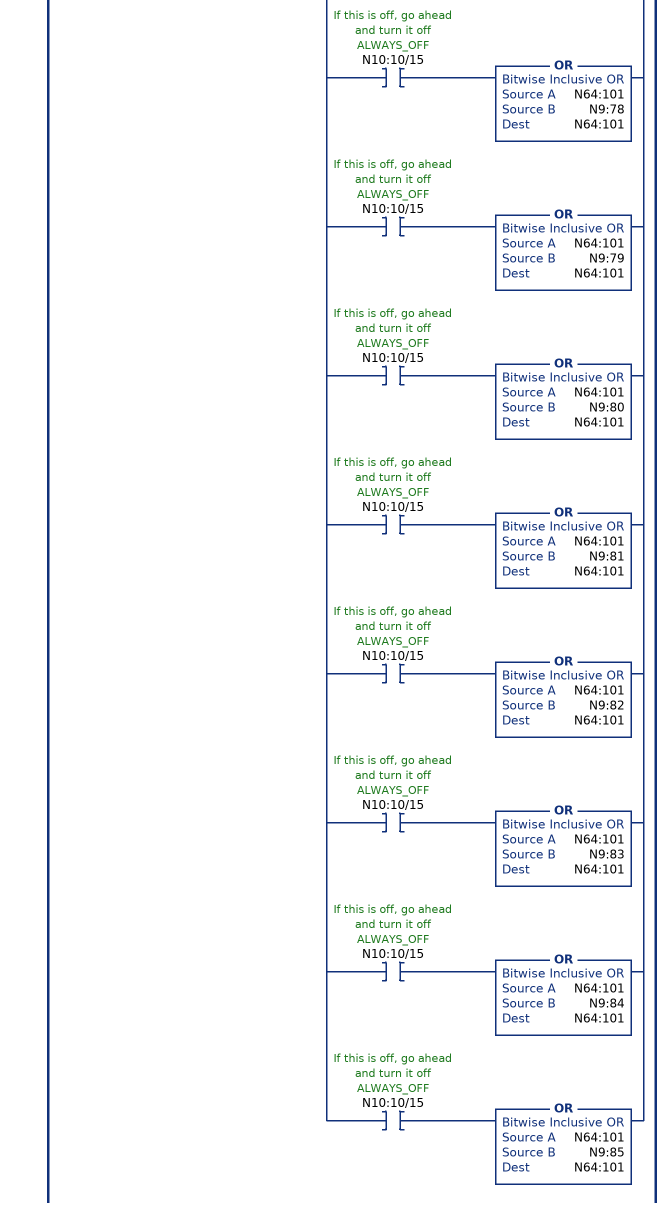
% Rung: 28 %
SOR EQU C5:19.ACC 11 XIO B3:0/3 BST MOV 0 N64:101 NXB XIC N10:10/15 OR N64:101 N9:70 N64:101 NXB XIC N10:10/15 OR N64:101 N9:71 N64:101 NXB XIC N10:10/15 OR N64:101 N9:72 N64:101 NXB XIC N10:10/15 OR N64:101 N9:73 N64:101 NXB XIC N10:10/15 OR N64:101 N9:74 N64:101 NXB XIC N10:10/15 OR N64:101 N9:75 N64:101 NXB XIC N10:10/15 OR N64:101 N9:76 N64:101 NXB XIC N10:10/15 OR N64:101 N9:77 N64:101 NXB XIC N10:10/15 OR N64:101 N9:78 N64:101 NXB XIC N10:10/15 OR N64:101 N9:79 N64:101 NXB XIC N10:10/15 OR N64:101 N9:80 N64:101 NXB XIC N10:10/15 OR N64:101 N9:81 N64:101 NXB XIC N10:10/15 OR N64:101 N9:82 N64:101 NXB XIC N10:10/15 OR N64:101 N9:83 N64:101 NXB XIC N10:10/15 OR N64:101 N9:84 N64:101 NXB XIC N10:10/15 OR N64:101 N9:85 N64:101 BND EOR
%   C5:19  MODBUS_COIL_CTR %
%   B3:0/3  MODBUS_TEST %
%   N10:10/15  ALWAYS_OFF  "If this is off, go ahead and turn it off" %
%   N9:70  BIT_0 %
%   N9:71  BIT_1 %
%   N9:72  BIT_2 %
%   N9:73  BIT_3 %
%   N9:74  BIT_4 %
%   N9:75  BIT_5 %
%   N9:76  BIT_6 %
%   N9:77  BIT_7 %
%   N9:78  BIT_8 %
%   N9:79  BIT_9 %
%   N9:80  BIT_10 %
%   N9:81  BIT_11 %
%   N9:82  BIT_12 %
%   N9:83  BIT_13 %
%   N9:84  BIT_14 %
%   N9:85  BIT_15 %

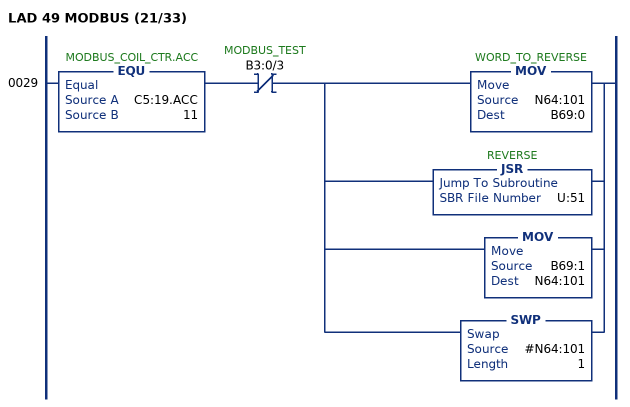
% Rung: 29 %
SOR EQU C5:19.ACC 11 XIO B3:0/3 BST MOV N64:101 B69:0 NXB JSR U:51 NXB MOV B69:1 N64:101 NXB SWP #N64:101 1 BND EOR
%   C5:19  MODBUS_COIL_CTR %
%   B3:0/3  MODBUS_TEST %
%   B69:0  WORD_TO_REVERSE %
%   U:51  REVERSE %
%   B69:1  REVERSED_WORD %

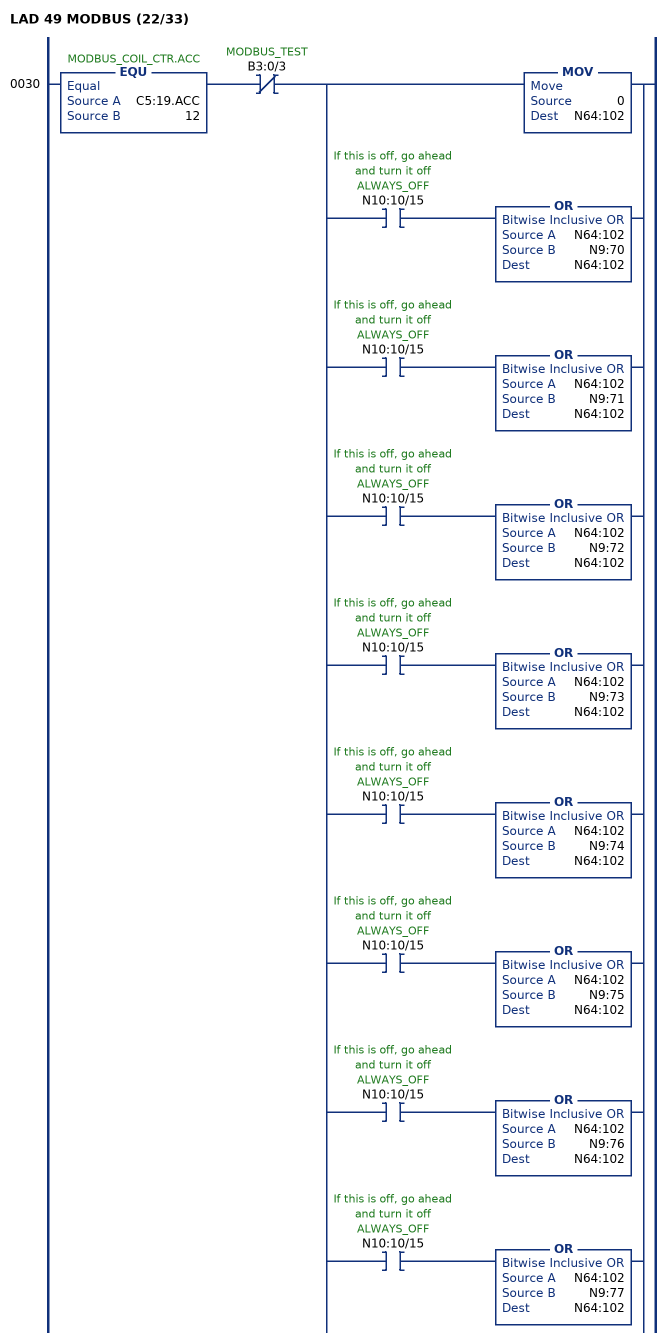

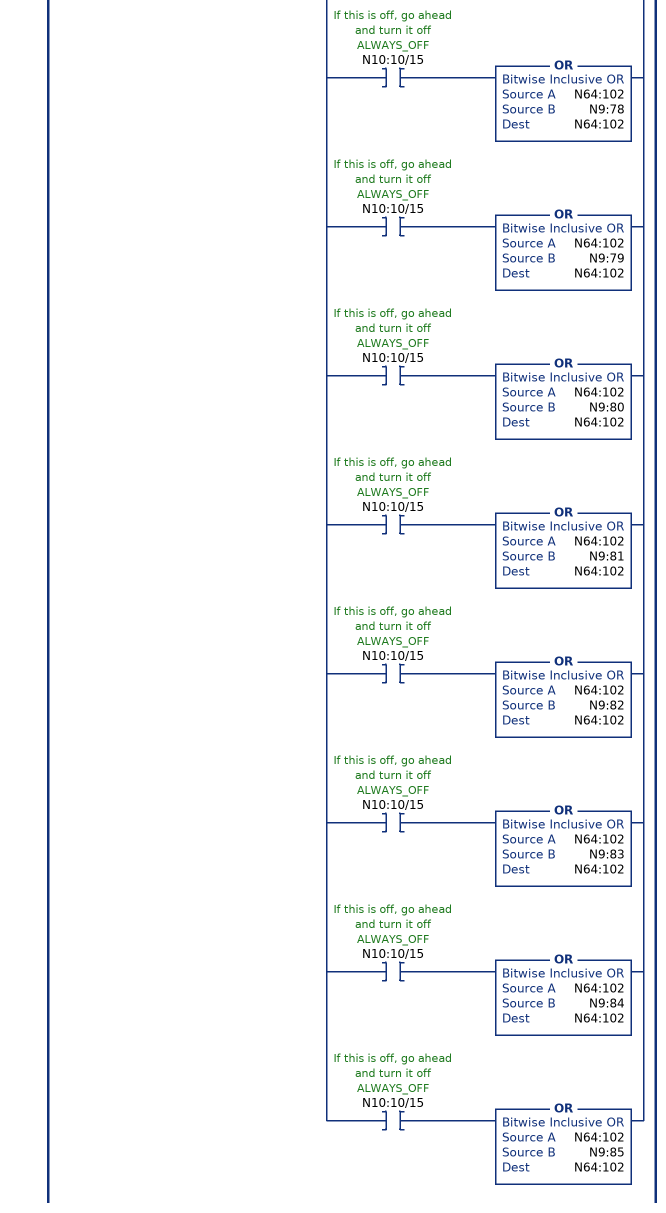
% Rung: 30 %
SOR EQU C5:19.ACC 12 XIO B3:0/3 BST MOV 0 N64:102 NXB XIC N10:10/15 OR N64:102 N9:70 N64:102 NXB XIC N10:10/15 OR N64:102 N9:71 N64:102 NXB XIC N10:10/15 OR N64:102 N9:72 N64:102 NXB XIC N10:10/15 OR N64:102 N9:73 N64:102 NXB XIC N10:10/15 OR N64:102 N9:74 N64:102 NXB XIC N10:10/15 OR N64:102 N9:75 N64:102 NXB XIC N10:10/15 OR N64:102 N9:76 N64:102 NXB XIC N10:10/15 OR N64:102 N9:77 N64:102 NXB XIC N10:10/15 OR N64:102 N9:78 N64:102 NXB XIC N10:10/15 OR N64:102 N9:79 N64:102 NXB XIC N10:10/15 OR N64:102 N9:80 N64:102 NXB XIC N10:10/15 OR N64:102 N9:81 N64:102 NXB XIC N10:10/15 OR N64:102 N9:82 N64:102 NXB XIC N10:10/15 OR N64:102 N9:83 N64:102 NXB XIC N10:10/15 OR N64:102 N9:84 N64:102 NXB XIC N10:10/15 OR N64:102 N9:85 N64:102 BND EOR
%   C5:19  MODBUS_COIL_CTR %
%   B3:0/3  MODBUS_TEST %
%   N10:10/15  ALWAYS_OFF  "If this is off, go ahead and turn it off" %
%   N9:70  BIT_0 %
%   N9:71  BIT_1 %
%   N9:72  BIT_2 %
%   N9:73  BIT_3 %
%   N9:74  BIT_4 %
%   N9:75  BIT_5 %
%   N9:76  BIT_6 %
%   N9:77  BIT_7 %
%   N9:78  BIT_8 %
%   N9:79  BIT_9 %
%   N9:80  BIT_10 %
%   N9:81  BIT_11 %
%   N9:82  BIT_12 %
%   N9:83  BIT_13 %
%   N9:84  BIT_14 %
%   N9:85  BIT_15 %

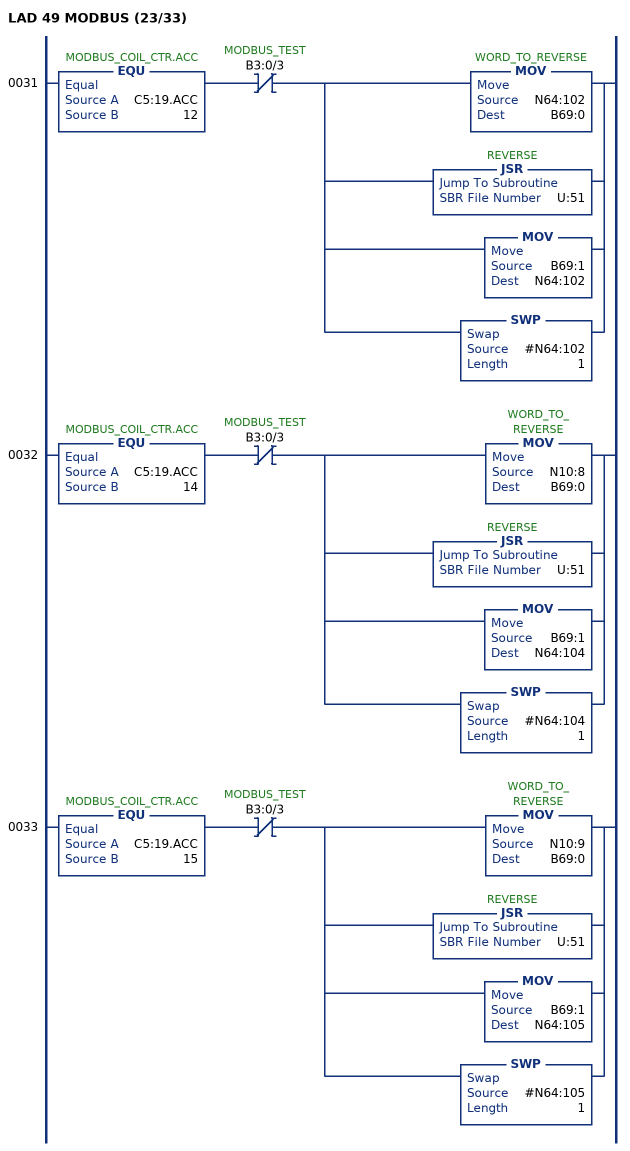
% Rung: 31 %
SOR EQU C5:19.ACC 12 XIO B3:0/3 BST MOV N64:102 B69:0 NXB JSR U:51 NXB MOV B69:1 N64:102 NXB SWP #N64:102 1 BND EOR
%   C5:19  MODBUS_COIL_CTR %
%   B3:0/3  MODBUS_TEST %
%   B69:0  WORD_TO_REVERSE %
%   U:51  REVERSE %
%   B69:1  REVERSED_WORD %
% Rung: 32 %
SOR EQU C5:19.ACC 14 XIO B3:0/3 BST MOV N10:8 B69:0 NXB JSR U:51 NXB MOV B69:1 N64:104 NXB SWP #N64:104 1 BND EOR
%   C5:19  MODBUS_COIL_CTR %
%   B3:0/3  MODBUS_TEST %
%   N10:8  SYSTEM_WARNINGS_0  "WARNING System Warnings" %
%   B69:0  WORD_TO_REVERSE %
%   U:51  REVERSE %
%   B69:1  REVERSED_WORD %
% Rung: 33 %
SOR EQU C5:19.ACC 15 XIO B3:0/3 BST MOV N10:9 B69:0 NXB JSR U:51 NXB MOV B69:1 N64:105 NXB SWP #N64:105 1 BND EOR
%   C5:19  MODBUS_COIL_CTR %
%   B3:0/3  MODBUS_TEST %
%   N10:9  SYSTEM_WARNINGS_1  "WARNING System Warnings" %
%   B69:0  WORD_TO_REVERSE %
%   U:51  REVERSE %
%   B69:1  REVERSED_WORD %

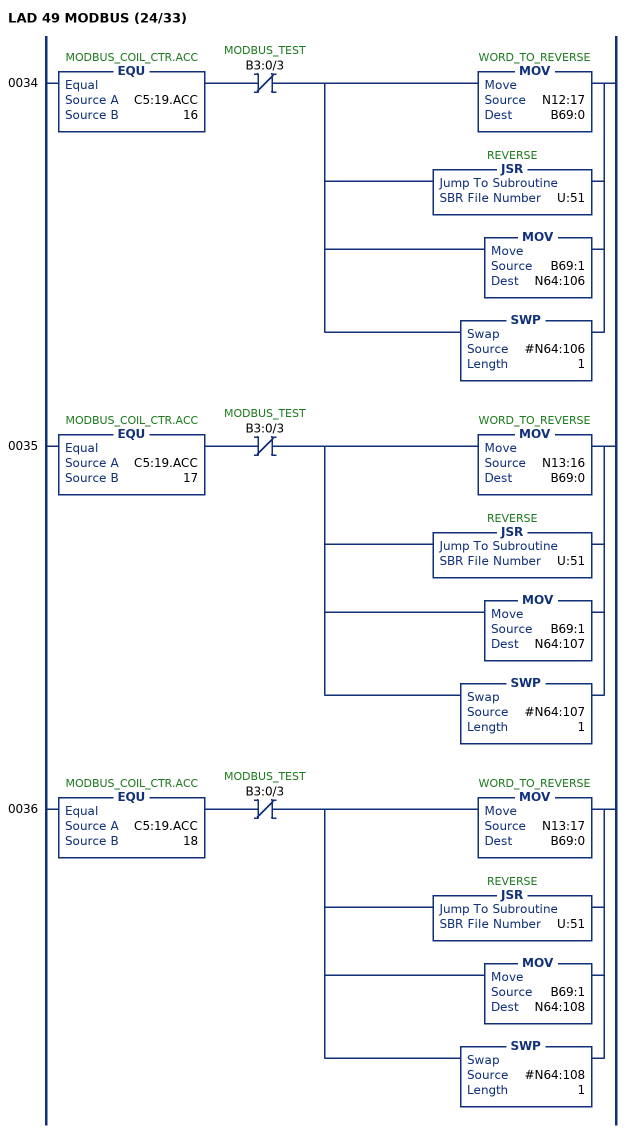
% Rung: 34 %
SOR EQU C5:19.ACC 16 XIO B3:0/3 BST MOV N12:17 B69:0 NXB JSR U:51 NXB MOV B69:1 N64:106 NXB SWP #N64:106 1 BND EOR
%   C5:19  MODBUS_COIL_CTR %
%   B3:0/3  MODBUS_TEST %
%   N12:17  PURIFY_WARNINGS_0 %
%   B69:0  WORD_TO_REVERSE %
%   U:51  REVERSE %
%   B69:1  REVERSED_WORD %
% Rung: 35 %
SOR EQU C5:19.ACC 17 XIO B3:0/3 BST MOV N13:16 B69:0 NXB JSR U:51 NXB MOV B69:1 N64:107 NXB SWP #N64:107 1 BND EOR
%   C5:19  MODBUS_COIL_CTR %
%   B3:0/3  MODBUS_TEST %
%   N13:16  REGEN_WARNINGS_0 %
%   B69:0  WORD_TO_REVERSE %
%   U:51  REVERSE %
%   B69:1  REVERSED_WORD %
% Rung: 36 %
SOR EQU C5:19.ACC 18 XIO B3:0/3 BST MOV N13:17 B69:0 NXB JSR U:51 NXB MOV B69:1 N64:108 NXB SWP #N64:108 1 BND EOR
%   C5:19  MODBUS_COIL_CTR %
%   B3:0/3  MODBUS_TEST %
%   N13:17  REGEN_WARNINGS_1 %
%   B69:0  WORD_TO_REVERSE %
%   U:51  REVERSE %
%   B69:1  REVERSED_WORD %

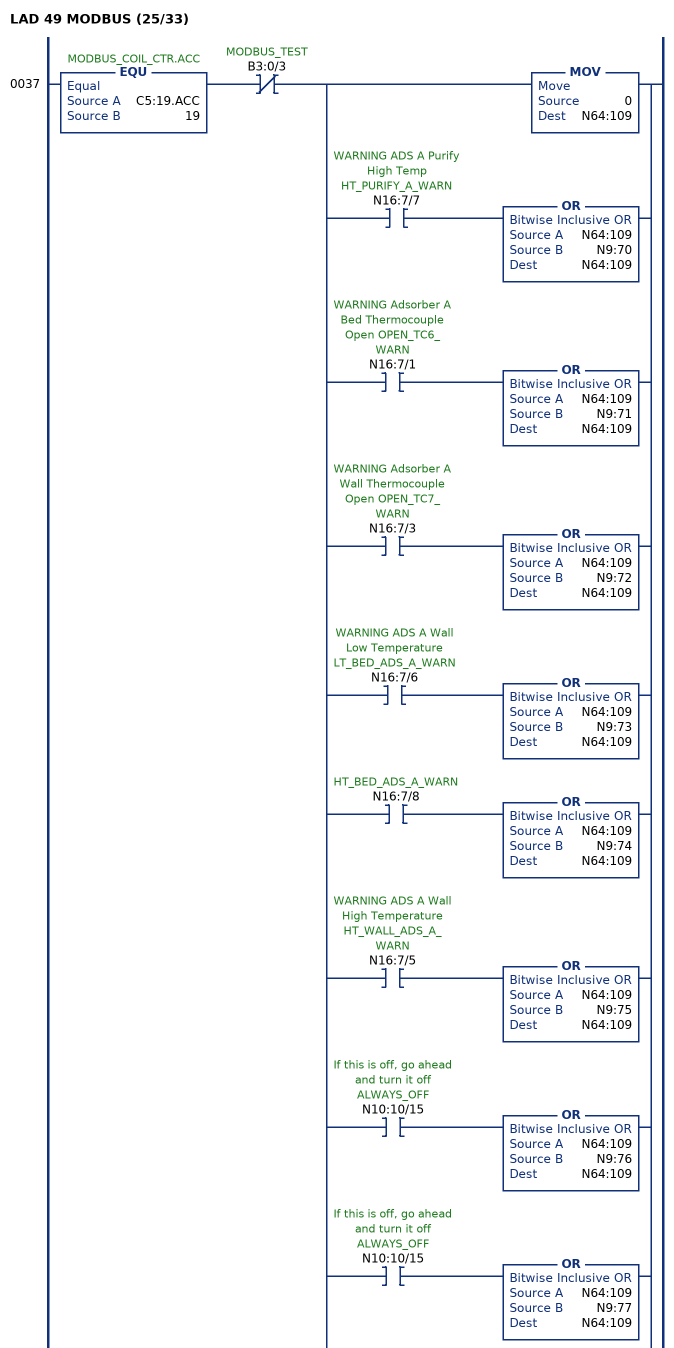

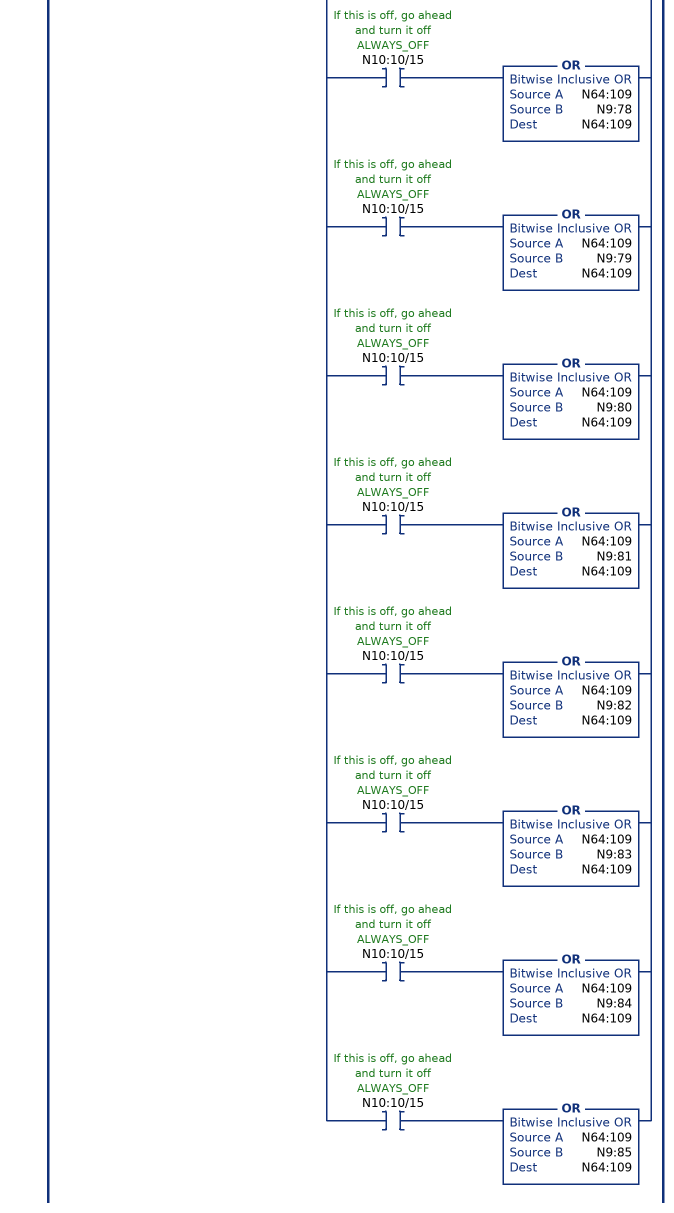
% Rung: 37 %
SOR EQU C5:19.ACC 19 XIO B3:0/3 BST MOV 0 N64:109 NXB XIC N16:7/7 OR N64:109 N9:70 N64:109 NXB XIC N16:7/1 OR N64:109 N9:71 N64:109 NXB XIC N16:7/3 OR N64:109 N9:72 N64:109 NXB XIC N16:7/6 OR N64:109 N9:73 N64:109 NXB XIC N16:7/8 OR N64:109 N9:74 N64:109 NXB XIC N16:7/5 OR N64:109 N9:75 N64:109 NXB XIC N10:10/15 OR N64:109 N9:76 N64:109 NXB XIC N10:10/15 OR N64:109 N9:77 N64:109 NXB XIC N10:10/15 OR N64:109 N9:78 N64:109 NXB XIC N10:10/15 OR N64:109 N9:79 N64:109 NXB XIC N10:10/15 OR N64:109 N9:80 N64:109 NXB XIC N10:10/15 OR N64:109 N9:81 N64:109 NXB XIC N10:10/15 OR N64:109 N9:82 N64:109 NXB XIC N10:10/15 OR N64:109 N9:83 N64:109 NXB XIC N10:10/15 OR N64:109 N9:84 N64:109 NXB XIC N10:10/15 OR N64:109 N9:85 N64:109 BND EOR
%   C5:19  MODBUS_COIL_CTR %
%   B3:0/3  MODBUS_TEST %
%   N16:7/7  HT_PURIFY_A_WARN  "WARNING ADS A Purify High Temp" %
%   N9:70  BIT_0 %
%   N16:7/1  OPEN_TC6_WARN  "WARNING Adsorber A Bed Thermocouple Open" %
%   N9:71  BIT_1 %
%   N16:7/3  OPEN_TC7_WARN  "WARNING Adsorber A Wall Thermocouple Open" %
%   N9:72  BIT_2 %
%   N16:7/6  LT_BED_ADS_A_WARN  "WARNING ADS A Wall Low Temperature" %
%   N9:73  BIT_3 %
%   N16:7/8  HT_BED_ADS_A_WARN %
%   N9:74  BIT_4 %
%   N16:7/5  HT_WALL_ADS_A_WARN  "WARNING ADS A Wall High Temperature" %
%   N9:75  BIT_5 %
%   N10:10/15  ALWAYS_OFF  "If this is off, go ahead and turn it off" %
%   N9:76  BIT_6 %
%   N9:77  BIT_7 %
%   N9:78  BIT_8 %
%   N9:79  BIT_9 %
%   N9:80  BIT_10 %
%   N9:81  BIT_11 %
%   N9:82  BIT_12 %
%   N9:83  BIT_13 %
%   N9:84  BIT_14 %
%   N9:85  BIT_15 %

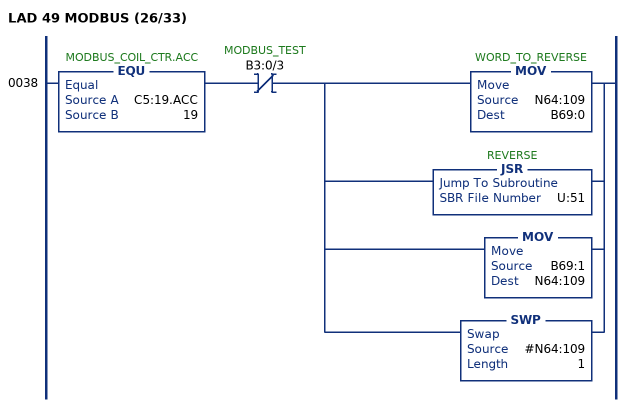
% Rung: 38 %
SOR EQU C5:19.ACC 19 XIO B3:0/3 BST MOV N64:109 B69:0 NXB JSR U:51 NXB MOV B69:1 N64:109 NXB SWP #N64:109 1 BND EOR
%   C5:19  MODBUS_COIL_CTR %
%   B3:0/3  MODBUS_TEST %
%   B69:0  WORD_TO_REVERSE %
%   U:51  REVERSE %
%   B69:1  REVERSED_WORD %

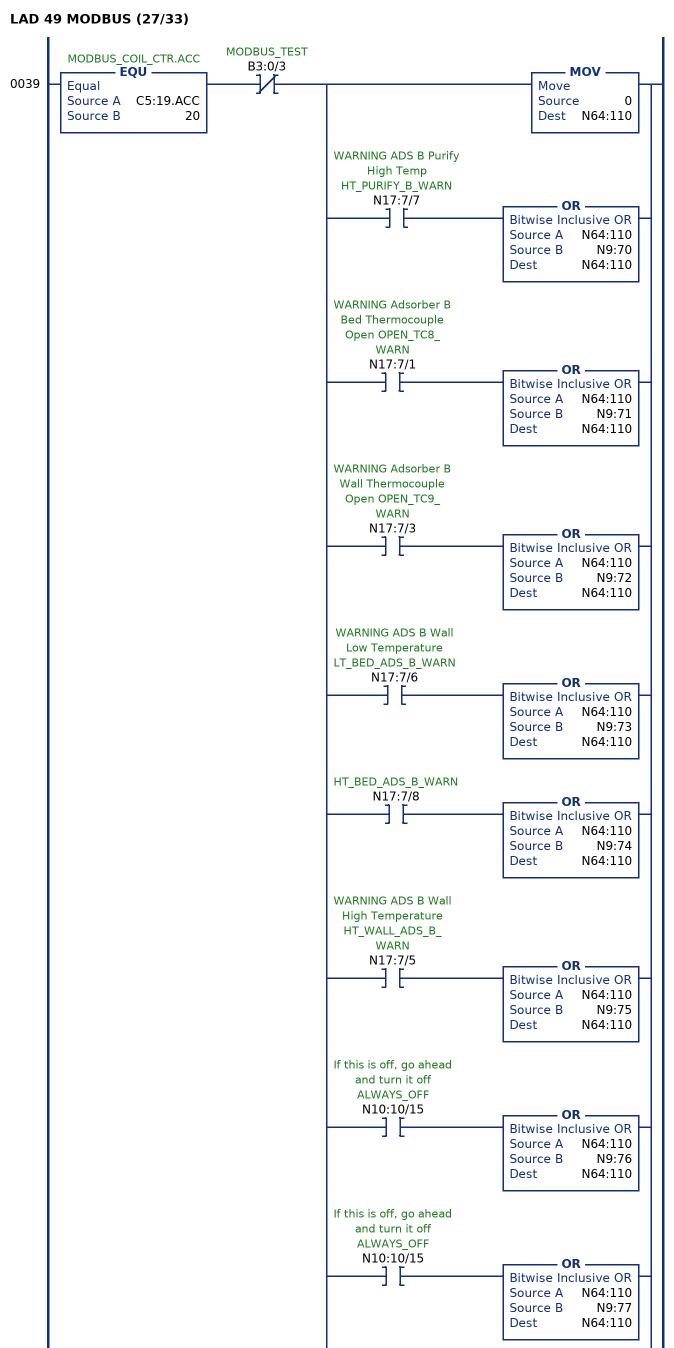

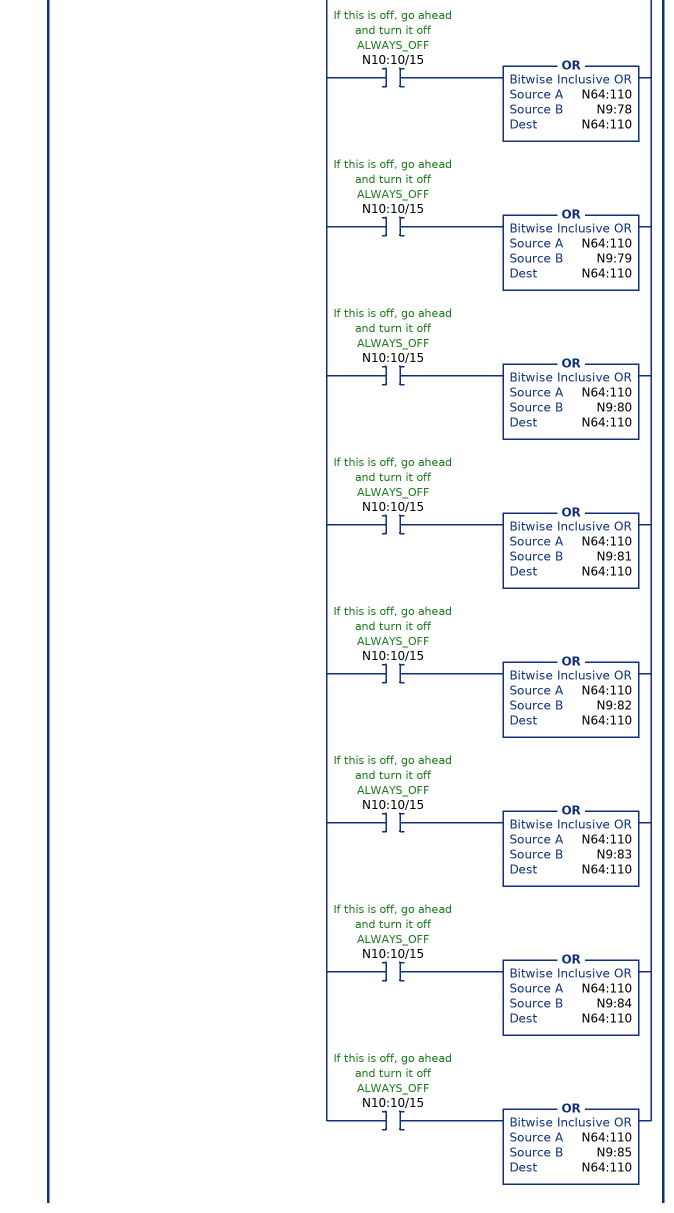
% Rung: 39 %
SOR EQU C5:19.ACC 20 XIO B3:0/3 BST MOV 0 N64:110 NXB XIC N17:7/7 OR N64:110 N9:70 N64:110 NXB XIC N17:7/1 OR N64:110 N9:71 N64:110 NXB XIC N17:7/3 OR N64:110 N9:72 N64:110 NXB XIC N17:7/6 OR N64:110 N9:73 N64:110 NXB XIC N17:7/8 OR N64:110 N9:74 N64:110 NXB XIC N17:7/5 OR N64:110 N9:75 N64:110 NXB XIC N10:10/15 OR N64:110 N9:76 N64:110 NXB XIC N10:10/15 OR N64:110 N9:77 N64:110 NXB XIC N10:10/15 OR N64:110 N9:78 N64:110 NXB XIC N10:10/15 OR N64:110 N9:79 N64:110 NXB XIC N10:10/15 OR N64:110 N9:80 N64:110 NXB XIC N10:10/15 OR N64:110 N9:81 N64:110 NXB XIC N10:10/15 OR N64:110 N9:82 N64:110 NXB XIC N10:10/15 OR N64:110 N9:83 N64:110 NXB XIC N10:10/15 OR N64:110 N9:84 N64:110 NXB XIC N10:10/15 OR N64:110 N9:85 N64:110 BND EOR
%   C5:19  MODBUS_COIL_CTR %
%   B3:0/3  MODBUS_TEST %
%   N17:7/7  HT_PURIFY_B_WARN  "WARNING ADS B Purify High Temp" %
%   N9:70  BIT_0 %
%   N17:7/1  OPEN_TC8_WARN  "WARNING Adsorber B Bed Thermocouple Open" %
%   N9:71  BIT_1 %
%   N17:7/3  OPEN_TC9_WARN  "WARNING Adsorber B Wall Thermocouple Open" %
%   N9:72  BIT_2 %
%   N17:7/6  LT_BED_ADS_B_WARN  "WARNING ADS B Wall Low Temperature" %
%   N9:73  BIT_3 %
%   N17:7/8  HT_BED_ADS_B_WARN %
%   N9:74  BIT_4 %
%   N17:7/5  HT_WALL_ADS_B_WARN  "WARNING ADS B Wall High Temperature" %
%   N9:75  BIT_5 %
%   N10:10/15  ALWAYS_OFF  "If this is off, go ahead and turn it off" %
%   N9:76  BIT_6 %
%   N9:77  BIT_7 %
%   N9:78  BIT_8 %
%   N9:79  BIT_9 %
%   N9:80  BIT_10 %
%   N9:81  BIT_11 %
%   N9:82  BIT_12 %
%   N9:83  BIT_13 %
%   N9:84  BIT_14 %
%   N9:85  BIT_15 %

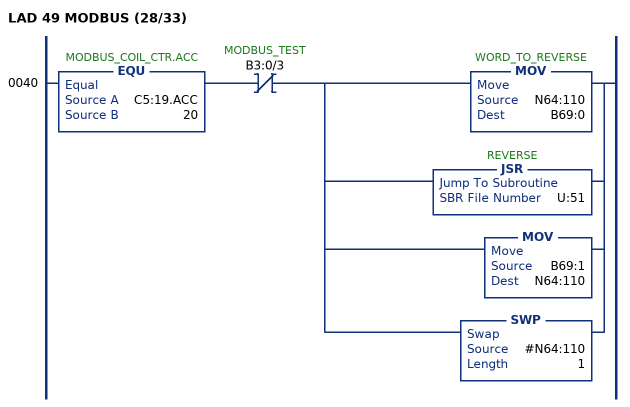
% Rung: 40 %
SOR EQU C5:19.ACC 20 XIO B3:0/3 BST MOV N64:110 B69:0 NXB JSR U:51 NXB MOV B69:1 N64:110 NXB SWP #N64:110 1 BND EOR
%   C5:19  MODBUS_COIL_CTR %
%   B3:0/3  MODBUS_TEST %
%   B69:0  WORD_TO_REVERSE %
%   U:51  REVERSE %
%   B69:1  REVERSED_WORD %

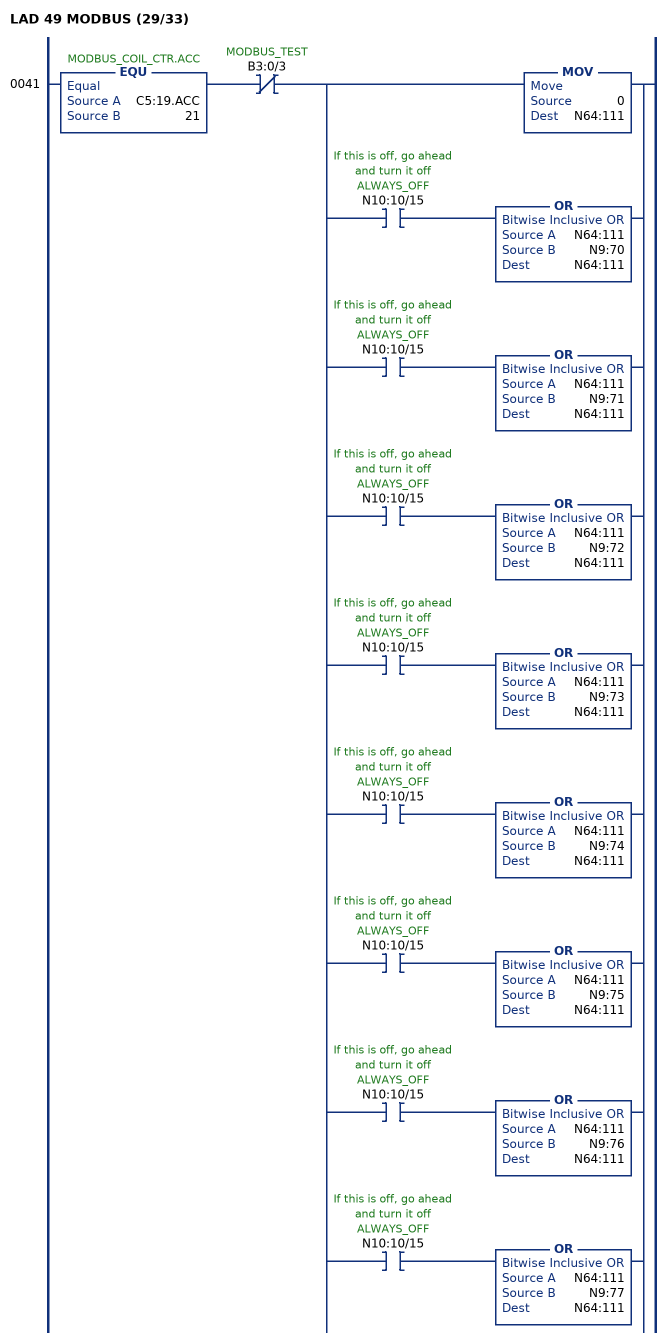

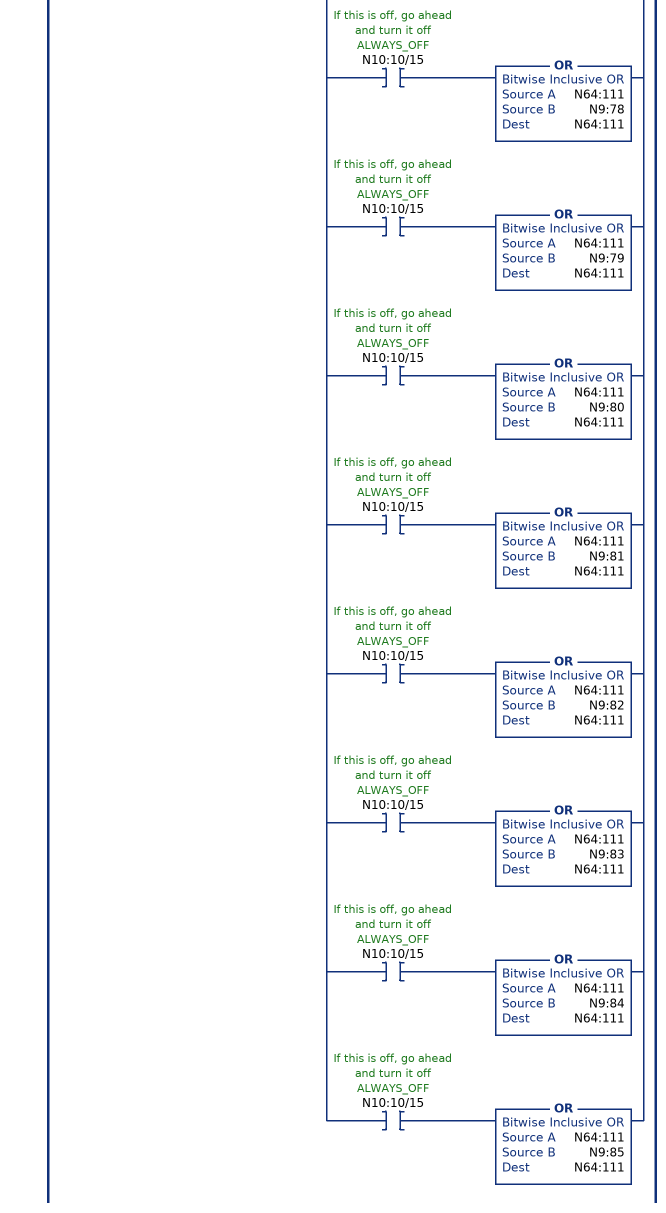
% Rung: 41 %
SOR EQU C5:19.ACC 21 XIO B3:0/3 BST MOV 0 N64:111 NXB XIC N10:10/15 OR N64:111 N9:70 N64:111 NXB XIC N10:10/15 OR N64:111 N9:71 N64:111 NXB XIC N10:10/15 OR N64:111 N9:72 N64:111 NXB XIC N10:10/15 OR N64:111 N9:73 N64:111 NXB XIC N10:10/15 OR N64:111 N9:74 N64:111 NXB XIC N10:10/15 OR N64:111 N9:75 N64:111 NXB XIC N10:10/15 OR N64:111 N9:76 N64:111 NXB XIC N10:10/15 OR N64:111 N9:77 N64:111 NXB XIC N10:10/15 OR N64:111 N9:78 N64:111 NXB XIC N10:10/15 OR N64:111 N9:79 N64:111 NXB XIC N10:10/15 OR N64:111 N9:80 N64:111 NXB XIC N10:10/15 OR N64:111 N9:81 N64:111 NXB XIC N10:10/15 OR N64:111 N9:82 N64:111 NXB XIC N10:10/15 OR N64:111 N9:83 N64:111 NXB XIC N10:10/15 OR N64:111 N9:84 N64:111 NXB XIC N10:10/15 OR N64:111 N9:85 N64:111 BND EOR
%   C5:19  MODBUS_COIL_CTR %
%   B3:0/3  MODBUS_TEST %
%   N10:10/15  ALWAYS_OFF  "If this is off, go ahead and turn it off" %
%   N9:70  BIT_0 %
%   N9:71  BIT_1 %
%   N9:72  BIT_2 %
%   N9:73  BIT_3 %
%   N9:74  BIT_4 %
%   N9:75  BIT_5 %
%   N9:76  BIT_6 %
%   N9:77  BIT_7 %
%   N9:78  BIT_8 %
%   N9:79  BIT_9 %
%   N9:80  BIT_10 %
%   N9:81  BIT_11 %
%   N9:82  BIT_12 %
%   N9:83  BIT_13 %
%   N9:84  BIT_14 %
%   N9:85  BIT_15 %

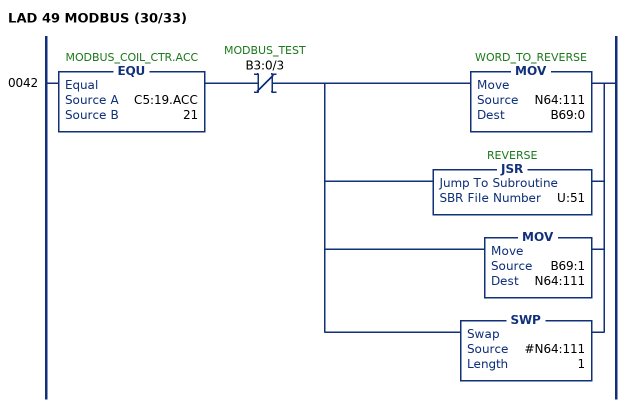
% Rung: 42 %
SOR EQU C5:19.ACC 21 XIO B3:0/3 BST MOV N64:111 B69:0 NXB JSR U:51 NXB MOV B69:1 N64:111 NXB SWP #N64:111 1 BND EOR
%   C5:19  MODBUS_COIL_CTR %
%   B3:0/3  MODBUS_TEST %
%   B69:0  WORD_TO_REVERSE %
%   U:51  REVERSE %
%   B69:1  REVERSED_WORD %

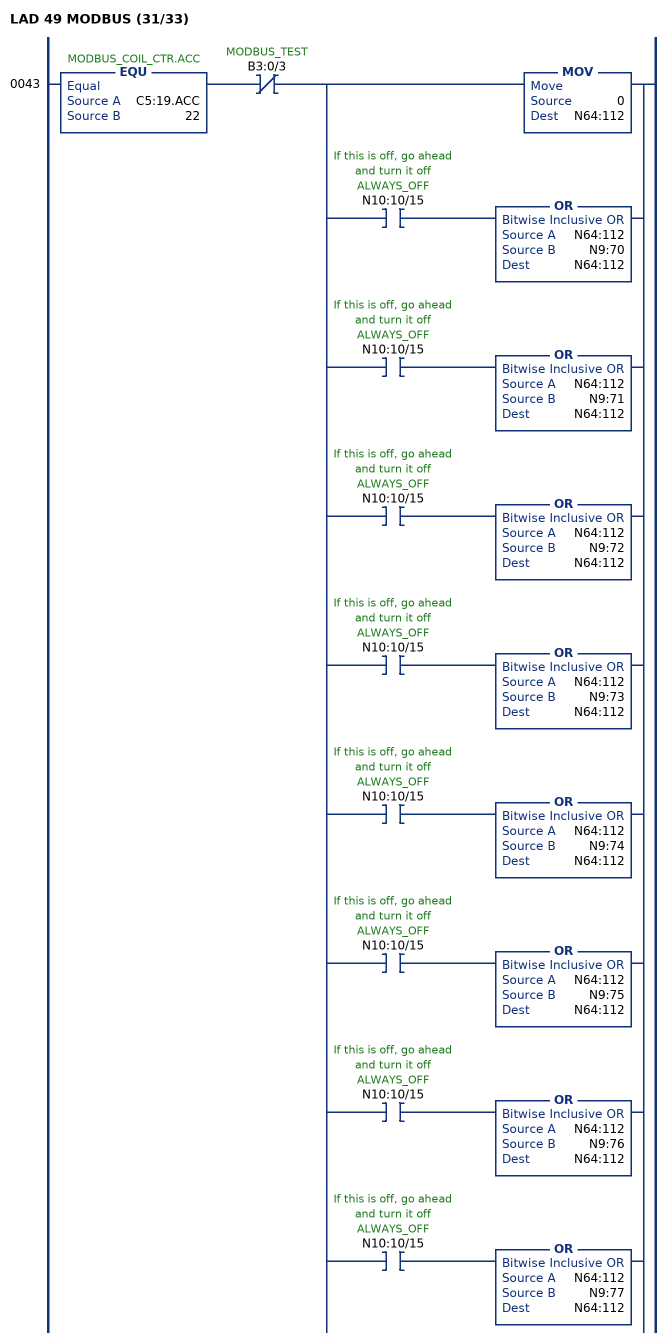

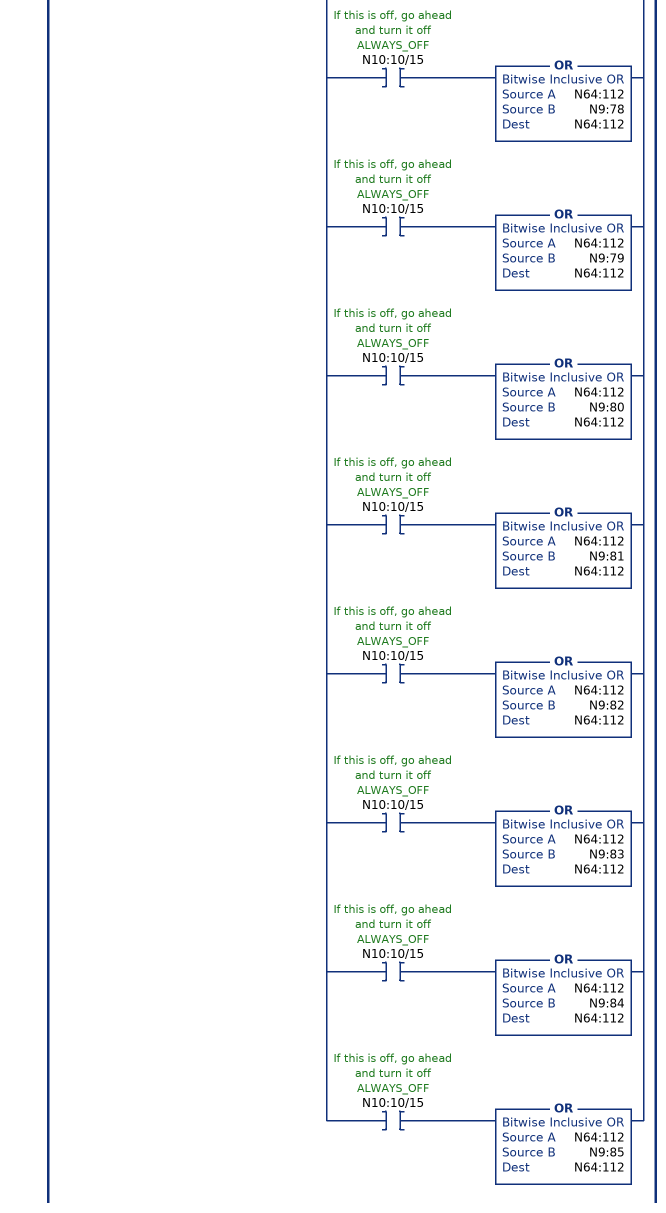
% Rung: 43 %
SOR EQU C5:19.ACC 22 XIO B3:0/3 BST MOV 0 N64:112 NXB XIC N10:10/15 OR N64:112 N9:70 N64:112 NXB XIC N10:10/15 OR N64:112 N9:71 N64:112 NXB XIC N10:10/15 OR N64:112 N9:72 N64:112 NXB XIC N10:10/15 OR N64:112 N9:73 N64:112 NXB XIC N10:10/15 OR N64:112 N9:74 N64:112 NXB XIC N10:10/15 OR N64:112 N9:75 N64:112 NXB XIC N10:10/15 OR N64:112 N9:76 N64:112 NXB XIC N10:10/15 OR N64:112 N9:77 N64:112 NXB XIC N10:10/15 OR N64:112 N9:78 N64:112 NXB XIC N10:10/15 OR N64:112 N9:79 N64:112 NXB XIC N10:10/15 OR N64:112 N9:80 N64:112 NXB XIC N10:10/15 OR N64:112 N9:81 N64:112 NXB XIC N10:10/15 OR N64:112 N9:82 N64:112 NXB XIC N10:10/15 OR N64:112 N9:83 N64:112 NXB XIC N10:10/15 OR N64:112 N9:84 N64:112 NXB XIC N10:10/15 OR N64:112 N9:85 N64:112 BND EOR
%   C5:19  MODBUS_COIL_CTR %
%   B3:0/3  MODBUS_TEST %
%   N10:10/15  ALWAYS_OFF  "If this is off, go ahead and turn it off" %
%   N9:70  BIT_0 %
%   N9:71  BIT_1 %
%   N9:72  BIT_2 %
%   N9:73  BIT_3 %
%   N9:74  BIT_4 %
%   N9:75  BIT_5 %
%   N9:76  BIT_6 %
%   N9:77  BIT_7 %
%   N9:78  BIT_8 %
%   N9:79  BIT_9 %
%   N9:80  BIT_10 %
%   N9:81  BIT_11 %
%   N9:82  BIT_12 %
%   N9:83  BIT_13 %
%   N9:84  BIT_14 %
%   N9:85  BIT_15 %

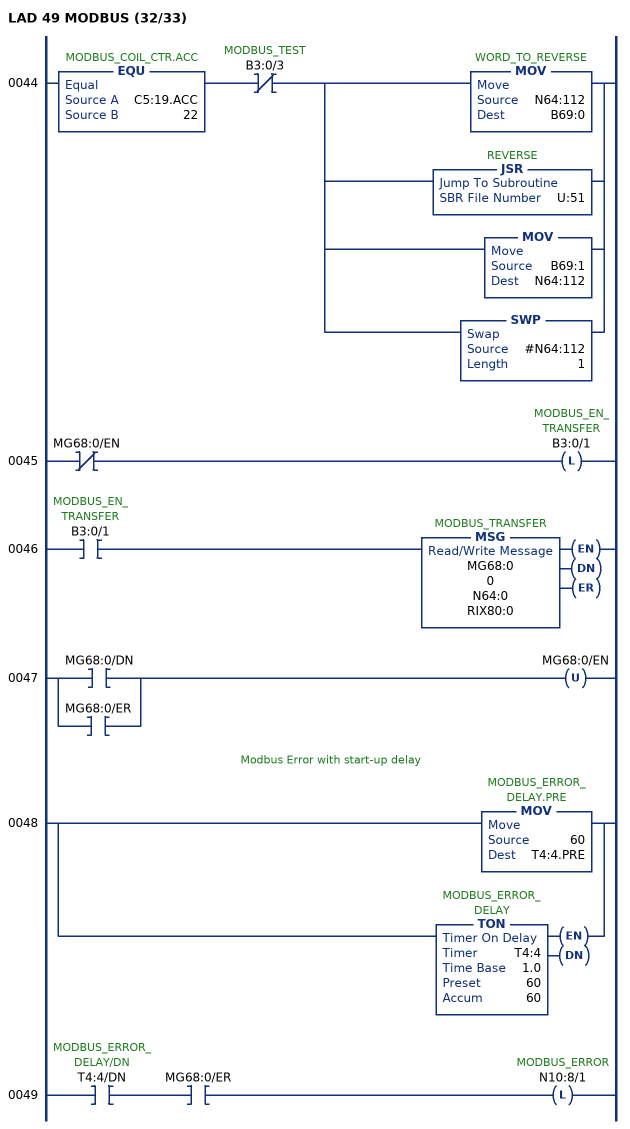
% Rung: 44 %
SOR EQU C5:19.ACC 22 XIO B3:0/3 BST MOV N64:112 B69:0 NXB JSR U:51 NXB MOV B69:1 N64:112 NXB SWP #N64:112 1 BND EOR
%   C5:19  MODBUS_COIL_CTR %
%   B3:0/3  MODBUS_TEST %
%   B69:0  WORD_TO_REVERSE %
%   U:51  REVERSE %
%   B69:1  REVERSED_WORD %
% Rung: 45 %
SOR XIO MG68:0/EN OTL B3:0/1 EOR
%   B3:0/1  MODBUS_EN_TRANSFER %
% Rung: 46 %
SOR XIC B3:0/1 MSG MG68:0 0 N64:0 RIX80:0 EOR
%   B3:0/1  MODBUS_EN_TRANSFER %
%   MSG set-up: CIP Generic | 33 | 0 | ? | 0 | 0 | 0 | 0 | 172.16.14.73:502 | 0 | 0 | 172.16.14.73 | RIX80:0 | 10 | 4 | 150 | 3 | 4 | 96 | 3 | 252 | N64:0 %
%   MG68:0  MODBUS_TRANSFER %
%   N64:0  REGISTER_START %
% Rung: 47 %
SOR BST XIC MG68:0/DN NXB XIC MG68:0/ER BND OTU MG68:0/EN EOR
% Rung: 48 %
% Modbus Error with start-up delay %
SOR BST MOV 60 T4:4.PRE NXB TON T4:4 1.0 60 60 BND EOR
%   T4:4  MODBUS_ERROR_DELAY %
% Rung: 49 %
SOR XIC T4:4/DN XIC MG68:0/ER OTL N10:8/1 EOR
%   T4:4  MODBUS_ERROR_DELAY %
%   N10:8/1  MODBUS_ERROR %

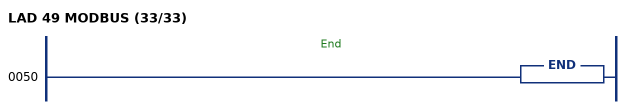
% Rung: 50 %
% End %
SOR END EOR

LADDER 50 "PLC_FAULT"
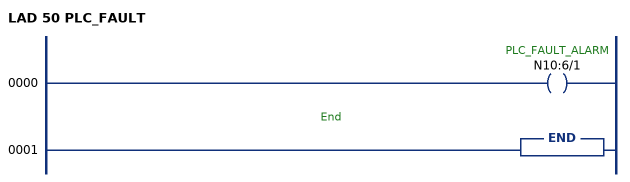
% Rung: 0 %
SOR OTE N10:6/1 EOR
%   N10:6/1  PLC_FAULT_ALARM %
% Rung: 1 %
% End %
SOR END EOR

LADDER 51 "REVERSE"
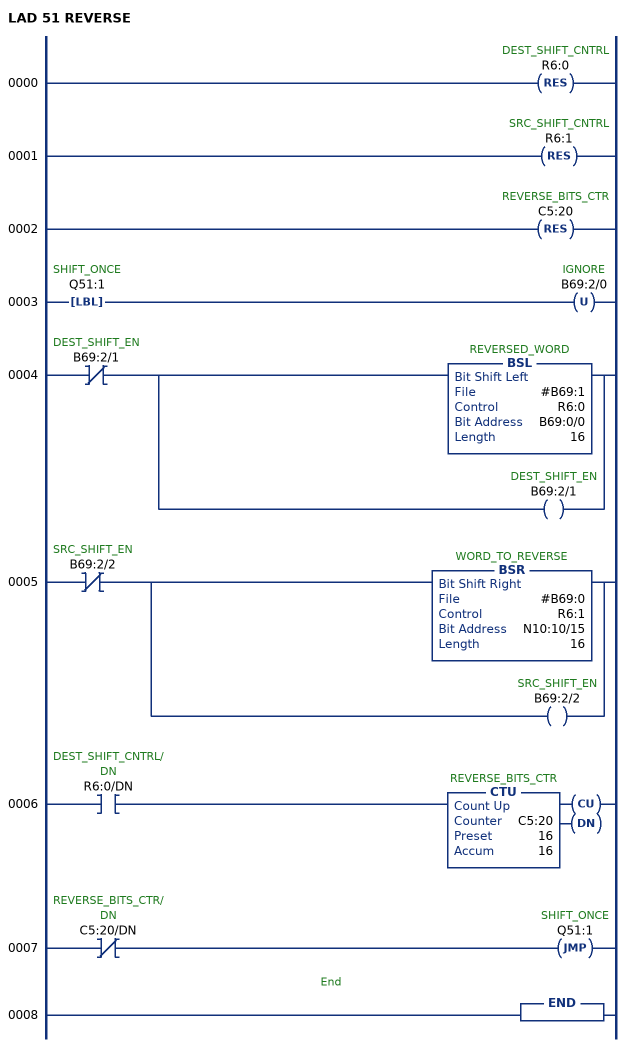
% Rung: 0 %
SOR RES R6:0 EOR
%   R6:0  DEST_SHIFT_CNTRL %
% Rung: 1 %
SOR RES R6:1 EOR
%   R6:1  SRC_SHIFT_CNTRL %
% Rung: 2 %
SOR RES C5:20 EOR
%   C5:20  REVERSE_BITS_CTR %
% Rung: 3 %
SOR LBL Q51:1 OTU B69:2/0 EOR
%   Q51:1  SHIFT_ONCE %
%   B69:2/0  IGNORE %
% Rung: 4 %
SOR XIO B69:2/1 BST BSL #B69:1 R6:0 B69:0/0 16 NXB OTE B69:2/1 BND EOR
%   B69:2/1  DEST_SHIFT_EN %
%   B69:1  REVERSED_WORD %
%   R6:0  DEST_SHIFT_CNTRL %
% Rung: 5 %
SOR XIO B69:2/2 BST BSR #B69:0 R6:1 N10:10/15 16 NXB OTE B69:2/2 BND EOR
%   B69:2/2  SRC_SHIFT_EN %
%   B69:0  WORD_TO_REVERSE %
%   R6:1  SRC_SHIFT_CNTRL %
%   N10:10/15  ALWAYS_OFF  "If this is off, go ahead and turn it off" %
% Rung: 6 %
SOR XIC R6:0/DN CTU C5:20 16 16 EOR
%   R6:0  DEST_SHIFT_CNTRL %
%   C5:20  REVERSE_BITS_CTR %
% Rung: 7 %
SOR XIO C5:20/DN JMP Q51:1 EOR
%   C5:20  REVERSE_BITS_CTR %
%   Q51:1  SHIFT_ONCE %
% Rung: 8 %
% End %
SOR END EOR

OTHER DOCUMENTED ADDRESSES
  B30:0  CONFIG_BITS_HARDWARE  "CONFIG Hardware options installed"
  B30:1/15  CUSTOM_HP_GAS_LIMITS
  B30:5  SYSTEM_STATUS_0  "STATUS System Status of system contro entities"
  B31:2  SYSTEM_HMI_CMD_0  "COMMAND HMI Commands"
  B31:3  SYSTEM_HMI_CMD_1  "COMMAND HMI Commands"
  B31:4  SYSTEM_HMI_CMD_2  "COMMAND HMI Commands"
  B31:5  SYSTEM_HMI_CMD_3
  B31:6  SYSTEM_HMI_CMD_4  "COMMAND HMI Commands"
  B31:7  SYSTEM_HMI_CMD_5  "COMMAND HMI Commands"
  B33:0  PURIFY_HMI_CMDS
  B33:0/1  DEF_PURIFY_MAX
  B34:0  REGEN_HMI_CMDS
  B34:2  REGEN_FLAGS
  B35:2  MANUAL_HMI_CMNDS_0
  DFILE:0  "OUTPUT"
  DFILE:1  "INPUT"
  DFILE:2  "STATUS"
  DFILE:3  "BINARY"
  DFILE:4  "TIMER"
  DFILE:5  "COUNTER"
  DFILE:6  "CONTROL"
  DFILE:7  "SYSTEM CFG Maintains the values that characterize t he system"
  DFILE:8  "FLOAT"
  DFILE:9  "CONSTANTS The collection of sy stem and subsystem c onstants"
  DFILE:10  "SYSTEM Contain the values f or system control"
  DFILE:11  "PROCESS Contains the values for the processing m achine"
  DFILE:12  "PURIFY Contains the values required for purify"
  DFILE:13  "REGEN Contains the values required for regen"
  DFILE:14  "BYPASS"
  DFILE:15  "MANUAL CTL Contains the data fo r the manual valve c ontrol"
  DFILE:16  "ADSORBER_A Contains the values for Adsorber A"
  DFILE:17  "ADSORBER_B Contains the values required for Adsorbe r B"
  DFILE:18  "STATUS_PRC"
  DFILE:19  "ADSORBER_D"
  DFILE:20  "MIX PANEL"
  DFILE:21  "OUTLET"
  DFILE:23  "MB_HRTBT"
  DFILE:25  "PID HEATER"
  DFILE:30  "SYSTEM CFG"
  DFILE:31  "SYSTEM"
  DFILE:32  "PROCESS"
  DFILE:33  "PURIFY"
  DFILE:34  "REGEN"
  DFILE:35  "MANUAL CTL"
  DFILE:38  "HEATERS"
  DFILE:51  "TOTAL_FLOW"
  DFILE:64  "MODBUS"
  DFILE:68  "TRANSFER"
  DFILE:69  "REVERSE"
  DFILE:80  "MSG_SETUP"
  DFILE:207  "STATUS_PRC"
  N7:0  CONFIG_BITS_ALM
  N7:1  CONFIG_BITS_ALM_O  "CONFIG System alarms enable"
  N7:2  CONFIG_BITS_ALM_1  "CONFIG System alarms enable"
  N7:3  CONFIG_BITS_WARN_0  "CONFIG System warnings enable"
  N7:4  CONFIG_BITS_WARN_1  "CONFIG System warnings enable"
  N7:5  CONFIG_BITS_WARN
  N7:6  CONFIG_OPEN_TC_ALM
  N7:7  CONFIG_OPEN_TC_WARN
  N10:10  SYSTEM_CONTROL  "CONTROL System Bits used to manipulate hardware"
  N10:16  SYSTEM_FLAGS_1
  N12:4  PURIFY_FLAGS_0  "STATUS Flags used by the purify process"
  N12:5  PURIFY_CONTROL  "CONTROL Control bits used by the purify process to change hardware states"
  N12:10  PURIFY_FACTOR  "CONFIG The percent output requested by the operator (percent)"
  N12:12  PURIFY_CALC_0  "CONFIG Math result placeholder for the purify time calculation"
  N12:13  PURIFY_FACTOR_TIME  "CONFIG The factored purify time accounting for the purify percent factor (hours)"
  N12:14  PURIFY_MAX_TIME
  N13:5  REGEN_CONTROL  "CONTROL Regen Bits used to manipulate hardware"
  N14:1  BYPASS_COMMAND
  N15:4  MANUAL_FLAGS_0
  N16:3  ADS_A_FLAGS_0  "STATUS Flags used for Adsorber A"
  N17:3  ADS_B_FLAGS_0  "STATUS Flags used for Adsorber B"
  T4:44  REG_RESUME_DLY_TMR

COMMENTS NOT ATTACHED TO A CURRENT RUNG
  N18:5/7: If the delay timer has completed, latch the alarm.
    If the operator acknowledges, reset it.
  N16:5/1: ADSORBER A VESSEL BED TC6 OPEN CIRCUIT / Alarm
  N7:8: Scale analog inputs / TODO: Do we need to add the ability to adjust the ammonia sensor scaling?
  N9:39: Set the value for Regen Equalize
  U:29: Call the routine to operate the Adsorber D fault control
  B34:1/3: If the state of this machine is REGEN and the regen process is calling for the heaters to operate, operate the heaters
  B34:1/2: If the state of this machine is REGEN and the regen process is calling for the heaters to operate, operate the heaters
  N13:14/12: ADS A Gas Temp Thermocouple alarm
    If the alarm conditions are met, latch the alarm.
    If the operator acknowledges, reset it.
  B34:1/1: If the state of this machine is REGEN and the regen process is calling for the heaters to operate, operate the heaters
  B34:1/0: If the state of this machine is REGEN and the regen process is calling for the heaters to operate, operate the heaters
  B34:3/0: Start REGEN on an EXOTHERMED bed after an EXOTHERM triggered bed swap.
  N7:4/13: Blend Gas Leak default
  N13:14/14: ADSORBER A PREHEATER GAS HIGH TEMP / Alarm
  N13:14/15: ADSORBER A PREHEATER ROD HIGH TEMP / Alarm
  T4:130: ADSORBER A PREHEATER GAS TC10 OPEN CIRCUIT / Alarm
  T4:132: ADSORBER A PREHEATER WALL TC11 OPEN CIRCUIT / Alarm
  T4:8: ADSORBER A HIGH TEMP PURIFY / Alarm
  T4:9: Warning
  N16:5/8: ADSORBER A HIGH TEMP BED / Alarm
  N16:5/5: ADSORBER A HIGH TEMP WALL / Alarm
  T4:16: ADSORBER A LOW TEMP BED / Alarm
  T4:17: Warning
  N16:5/3: ADSORBER A VESSEL WALL TC7 OPEN CIRCUIT / Alarm
  N13:15/1: ADSORBER B PREHEATER ROD HIGH TEMP / Alarm
  N13:15/0: ADSORBER B PREHEATER GAS HIGH TEMP / Alarm
  T4:136: ADSORBER B PREHEATER WALL TC13 OPEN CIRCUIT / Alarm
  T4:134: ADSORBER B PREHEATER GAS TC12 OPEN CIRCUIT / Alarm
  N17:5/3: ADSORBER B VESSEL WALL TC9 OPEN CIRCUIT / Alarm
  N17:5/1: ADSORBER B VESSEL BED TC8 OPEN CIRCUIT / Alarm
  T4:19: Warning
  T4:18: ADSORBER B LOW TEMP WALL / Alarm
  N17:5/5: ADSORBER B HIGH TEMP WALL / Alarm
  N17:5/8: ADSORBER B HIGH TEMP BED / Alarm
  T4:11: Warning
  T4:10: ADSORBER B HIGH TEMP PURIFY / Alarm
  C5:12: Reset High Regen Deviation Warning Counters
  T4:64: Blend Gas Leak Warning
  T4:62: High Pressure Blend Gas Warning
  T4:60: Low Pressure Blend Gas Warning
  PD25:3.2: If the state of this machine is REGEN and the regen process is calling for the heaters to operate, operate the heaters
  T4:30: PURIFY HOLD / Alarm
  T4:36: HIGH OUTLET PRESSURE / Alarm
  T4:34: HIGH INLET PRESSURE / Alarm
  T4:32: LOW OUTLET GAS PRESSURE / Alarm
  T4:112: LOW INLET GAS PRESSURE / Alarm
  N12:15/0: PURIFY HOLD / Alarm
  N10:7/4: SAFETY VENT SWITCH / Alarm and Warning
  T4:42: GAS OUTLET PRESSURE XDUCER OPEN CIRCUIT / Alarm
  T4:40: GAS INLET PRESSURE XDUCER OPEN CIRCUIT / Alarm
  T4:72: PURIFY FAULTS / Inlet Gas Low Temp Alarm
  T4:52: HIGH TEMP INTERLOCKS / Alarm
  T4:38: LOW EXTERNAL PNEUMATIC PRESSURE / Alarm
  T4:78: LOW INTERNAL PNEUMATIC PRESSURE / Alarm
  T4:95: SYSTEM HARDWARE / EMO ENABLE TIMER - Delay enabling of EMO for 5 seconds during startup to eliminate spurious EMO activation which will pur purifier offline (SW2031_E/ 20 May 2015)

REVISION NOTES
  0: moved some bits out of N7 into B30
  1: moved bits out of N10 into B31
  2: moved bits from N15 into B35
  3: added the final data files. didn't need to move any bits
  4: updated configuration for TC and AI cards. updated DO module point assignments
  5: added logic for double-acting purify valves
  6: added rod and blanket limits
  7: added tags for default buttons
  8: cleaning up bed b pid control code
  9: removed h2 sensor and moved moisture sensor to channel 6
  10: changed processor name
  11: added px3 reading
  12: added call to mix panel routine
  13: test ok
  14: trying to clear plc fault by entering new pid default parameters
  15: changed stored PID values so that it maybe doesn't fault the PLC
  16: copid in new PID values from PS21
  17: cleared out the data table
  18: changed ADS_TC_OPEN_SP to 13700 by default
  19: setting default PID parameters
  20: added in preheater and blanket setpoints
  21: lots of changes to PID control
  22: fixed up PID defaults
  23: done testing
  24: got rid of separate PID defaults
  25: fixed loop update time bug in preheater defaults
  26: PID control done
  27: ok, now it's done. made Adsorber B use the same PID parameters as Adsorber A.
  28: added control for AV11 to system routine
  29: moved mixing panel valves into mixing panel routine
  30: some small fixes to the processing subroutine.
  31: cleaned up manual valve control for AV10, 11
  32: minor edit to purify factor calculation
  33: made some fixes to ADS_A routine including adding another state buffer for adsorber-only alarms.
  34: fixed up ADS_B routine so that it's like ADS_B
  35: Regen sequence modified and default regen paramters added
  36: added regen default comments
  37: added regen steps to constants
  38: Regen counter condition resets added
  39: Fixed regen standby buffer
  40: Regen buffering and sequencing checked and fixed
  41: Merged
  42: remove alarm aknowledge
  43: Updated alarm tag names
  44: PH fault changed
  45: manual mode PID taop PID control
  46: Added fail to cool alarm and warning
  47: trying to fix ph fault
  48: fixing open tc
  49: fixed open tc logic
  50: ok, now it's fixed

DATA TABLE (non-zero values as saved)
DATA T4
% .PRE .ACC %
% T4:0 % 60 0
% T4:1 % 60 34
% T4:2 % 6 0
% T4:3 % 60 0
% T4:4 % 60 60
% T4:5 % 60 0
% T4:6 % 1000 856
% T4:7 % 1000 864
% T4:8 % 5 0
% T4:9 % 5 0
% T4:10 % 5 0
% T4:11 % 5 0
% T4:12 % 5 0
% T4:13 % 60 0
% T4:14 % 60 26
% T4:15 % 60 0
% T4:16 % 21600 0
% T4:17 % 21600 0
% T4:18 % 21600 0
% T4:19 % 21600 0
% T4:20 % 5 0
% T4:21 % 60 0
% T4:22 % 5 0
% T4:23 % 60 0
% T4:24 % 1 0
% T4:25 % 1 0
% T4:26 % 5 0
% T4:27 % 5 0
% T4:28 % 5 0
% T4:29 % 5 0
% T4:30 % 60 0
% T4:31 % 60 0
% T4:32 % 5 0
% T4:33 % 5 0
% T4:34 % 5 0
% T4:35 % 5 0
% T4:36 % 5 0
% T4:37 % 5 0
% T4:38 % 5 0
% T4:39 % 60 0
% T4:40 % 5 0
% T4:41 % 5 0
% T4:42 % 5 0
% T4:43 % 5 0
% T4:44 % 2 0
% T4:46 % 5 0
% T4:47 % 5 0
% T4:48 % 5 0
% T4:49 % 60 0
% T4:50 % 5 0
% T4:51 % 60 0
% T4:52 % 2 0
% T4:53 % 2 0
% T4:54 % 500 103
% T4:55 % 60 0
% T4:56 % 60 0
% T4:57 % 30 0
% T4:58 % 30 0
% T4:59 % 5 0
% T4:60 % 5 0
% T4:61 % 10 0
% T4:62 % 10 0
% T4:63 % 60 0
% T4:64 % 60 0
% T4:65 % 60 3
% T4:66 % 60 0
% T4:67 % 60 0
% T4:68 % 60 0
% T4:69 % 60 26
% T4:70 % 5 0
% T4:71 % 5 0
% T4:72 % 5 0
% T4:73 % 5 0
% T4:74 % 60 0
% T4:75 % 60 0
% T4:76 % 5 0
% T4:77 % 60 0
% T4:78 % 5 0
% T4:79 % 5 0
% T4:80 % 5 0
% T4:81 % 5 0
% T4:83 % 5 0
% T4:85 % 5 0
% T4:87 % 5 0
% T4:88 % 5 0
% T4:89 % 5 0
% T4:90 % 21600 0
% T4:91 % 21600 0
% T4:92 % 21600 0
% T4:93 % 21600 0
% T4:94 % 5 5
% T4:95 % 500 0
% T4:97 % 5 0
% T4:98 % 60 0
% T4:99 % 5 0
% T4:100 % 5 0
% T4:101 % 5 0
% T4:102 % 5 0
% T4:105 % 5 0
% T4:106 % 60 0
% T4:111 % 60 0
% T4:112 % 5 0
% T4:113 % 5 0
% T4:114 % 60 0
% T4:117 % 60 0
% T4:120 % 60 0
% T4:121 % 60 10
% T4:122 % 5 0
% T4:123 % 5 0
% T4:124 % 5 0
% T4:126 % 5 0
% T4:127 % 5 0
% T4:128 % 5 0
% T4:130 % 5 0
% T4:132 % 5 0
% T4:134 % 5 0
% T4:136 % 5 0
% T4:142 % 5 0
% T4:143 % 5 0
% T4:146 % 5 0
% T4:147 % 5 0
% T4:148 % 5 0
% T4:149 % 5 0
% T4:150 % 5 0
% T4:151 % 5 0
% T4:152 % 5 0
% T4:153 % 5 0
DATA C5
% .PRE .ACC %
% C5:0 % 120 3
% C5:1 % 60 57
% C5:2 % 24 4
% C5:3 % 32767 0
% C5:4 % 1 0
% C5:5 % 180 0
% C5:7 % 10 0
% C5:8 % 1 0
% C5:9 % 5 1
% C5:10 % 5 0
% C5:11 % 5 0
% C5:12 % 5 0
% C5:13 % 30 126
% C5:14 % 10 0
% C5:15 % 600 126
% C5:17 % 800 0
% C5:18 % 800 0
% C5:19 % 23 1
% C5:20 % 16 16
% C5:21 % 60 0
% C5:22 % 1440 0
% C5:23 % 24 0
% C5:24 % 480 0
% C5:25 % 8 0
% C5:26 % 10 0
% C5:27 % 10 0
% C5:28 % 1 0
% C5:29 % 5 0
% C5:30 % 5 0
% C5:31 % 5 0
% C5:32 % 120 0
DATA R6
% .LEN .POS %
% R6:0 % 16 0
% R6:1 % 16 0
DATA T23
% .PRE .ACC %
% T23:1 % 100 62
% T23:2 % 100 0
DATA N64
% N64:0 % -12788 0 0 0 0 0 0 0 0 0
